FUNCTION_BLOCK DataTypesBitStrings (* Template for an empty basic function block *)
  (* Standard: 61499-2; Description: Normal just propagates the input to the output Internal: sets the output from inside Copyright (c) 2019 Jan Holzweber This program and the accompanying materials are made available under the terms of the Eclipse Public License 2.0 which is available at https://www.eclipse.org/legal/epl-2.0/ SPDX-License-Identifier: EPL-2.0 *)
  (* Version 1.0, 2019-06-05, jholz *)
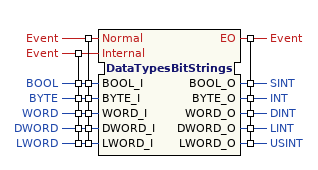
  EVENT_INPUT
    Normal WITH BOOL_I, WORD_I, DWORD_I, LWORD_I, BYTE_I;
    Internal WITH BOOL_I, WORD_I, DWORD_I, LWORD_I, BYTE_I;
  END_EVENT
  EVENT_OUTPUT
    EO WITH BOOL_O, BYTE_O, WORD_O, DWORD_O, LWORD_O;
  END_EVENT
  VAR_INPUT
    BOOL_I : BOOL;
    BYTE_I : BYTE;
    WORD_I : WORD;
    DWORD_I : DWORD;
    LWORD_I : LWORD;
  END_VAR
  VAR_OUTPUT
    BOOL_O : SINT;
    BYTE_O : INT;
    WORD_O : DINT;
    DWORD_O : LINT;
    LWORD_O : USINT;
  END_VAR
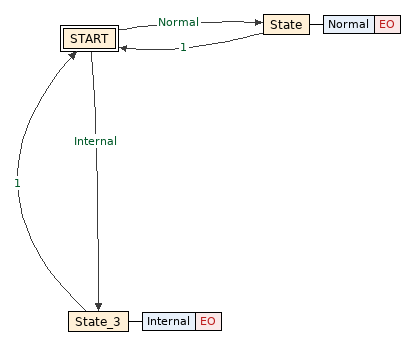
  EC_STATES
    START; (* Initial State *)
    State : Normal -> EO;
    State_3 : Internal -> EO;
  END_STATES
  EC_TRANSITIONS
    START TO State := Normal;
    State TO START := 1;
    START TO State_3 := Internal;
    State_3 TO START := 1;
  END_TRANSITIONS
  ALGORITHM Normal IN ST: (* new algorithm *)
BOOL_O:=BOOL_I;
BYTE_O:=BYTE_I;
WORD_O:=WORD_I;
DWORD_O:=DWORD_I;
LWORD_O:=LWORD_I;
  END_ALGORITHM
  ALGORITHM Internal IN ST: (* new algorithm *)
BOOL_O:=1;
BYTE_O:=2;
WORD_O:=35555;
DWORD_O:=2147483648;
LWORD_O:=2147483648;
  END_ALGORITHM
END_FUNCTION_BLOCK
